{attribute addProperty BoxType "EK1122-0000-0018"}
{attribute addProperty Id "Beckhoff_ER3xxxsub_EK1100EK1100_179A0949162A_0001_ER3174_0002_0016ER3174_83515A0D22428A_0002_ER3174_0002_0022ER3174_83515A0D22428A_0003_ER3174_0002_0023ER3174_83515A0D22428A_0004_ER3184_0002_0019ER3184_55F04E9922428A_0005_ER3184_0002_0020ER3184_55F04E9922428A_0006_ER3184_0002_0021ER3184_83515A0D22428A_0007_ER3184_1002_0020ER3184_55F04E9922428A_0008_ER3184_1002_0021ER3184_83515A0D22428A_0009_ER3204_0002_0016ER3204_BF093E1239249A_0010_ER3204_0002_0020ER3204_BF093E1239249A_0011_ER3204_0002_0021ER3204_69AA4F8E22428A_0012_ER3314_0002_0021ER3314_2E54E3B022428"}
{attribute addProperty CRC "3446871239"}
{attribute addProperty SizeInBites "3040"}
{attribute addProperty SizeInBytes "380"}
TYPE Beckhoff_ER3xxxEK1122_CD7314C7 EXTENDS EK1122_179A0949 :
STRUCT
	{attribute addProperty Name "Beckhoff_ER3xxxsub_EK1100"}
	Beckhoff_ER3xxxsub_EK1100 : EK1100_179A0949;
	{attribute addProperty Name "A_0001_ER3174_0002_0016"}
	A_0001_ER3174_0002_0016 : ER3174_83515A0D;
	{attribute addProperty Name "A_0002_ER3174_0002_0022"}
	A_0002_ER3174_0002_0022 : ER3174_83515A0D;
	{attribute addProperty Name "A_0003_ER3174_0002_0023"}
	A_0003_ER3174_0002_0023 : ER3174_83515A0D;
	{attribute addProperty Name "A_0004_ER3184_0002_0019"}
	A_0004_ER3184_0002_0019 : ER3184_55F04E99;
	{attribute addProperty Name "A_0005_ER3184_0002_0020"}
	A_0005_ER3184_0002_0020 : ER3184_55F04E99;
	{attribute addProperty Name "A_0006_ER3184_0002_0021"}
	A_0006_ER3184_0002_0021 : ER3184_83515A0D;
	{attribute addProperty Name "A_0007_ER3184_1002_0020"}
	A_0007_ER3184_1002_0020 : ER3184_55F04E99;
	{attribute addProperty Name "A_0008_ER3184_1002_0021"}
	A_0008_ER3184_1002_0021 : ER3184_83515A0D;
	{attribute addProperty Name "A_0009_ER3204_0002_0016"}
	A_0009_ER3204_0002_0016 : ER3204_BF093E12;
	{attribute addProperty Name "A_0010_ER3204_0002_0020"}
	A_0010_ER3204_0002_0020 : ER3204_BF093E12;
	{attribute addProperty Name "A_0011_ER3204_0002_0021"}
	A_0011_ER3204_0002_0021 : ER3204_69AA4F8E;
	{attribute addProperty Name "A_0012_ER3314_0002_0021"}
	A_0012_ER3314_0002_0021 : ER3314_2E54E3B0;
END_STRUCT
END_TYPE

(* stored: Version 1.2.0.0, ProductVersion 3.1.4024.9
   DUT Beckhoff_ER3xxxEK1122_CD7314C7: Id {5898575f-05ed-461f-baca-5dde46c4a9a3} *)
